TYPE SimpleRelayProcesses :
STRUCT
	///Set the relay enabled or disabled
	setEnabled: SetEnabledProcess;
END_STRUCT
END_TYPE

(* stored: Version 1.1.0.1, ProductVersion 3.1.4019.2
   DUT SimpleRelayProcesses: Id {24dbf0fc-a78d-40c7-b324-ea2d46fc3dfc} *)
